FUNCTION_BLOCK PreTratamentoPreliminar (* Composite Function Block Type *)
  (* Standard: 61499-2 *)
  (* Version 0.0, 11/03/2026, template *)
  PACKAGE Hidryco.HidrycoLib;
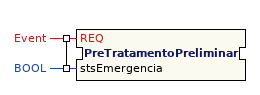
  EVENT_INPUT
    REQ WITH stsEmergencia;
  END_EVENT
  VAR_INPUT
    stsEmergencia : BOOL;
  END_VAR
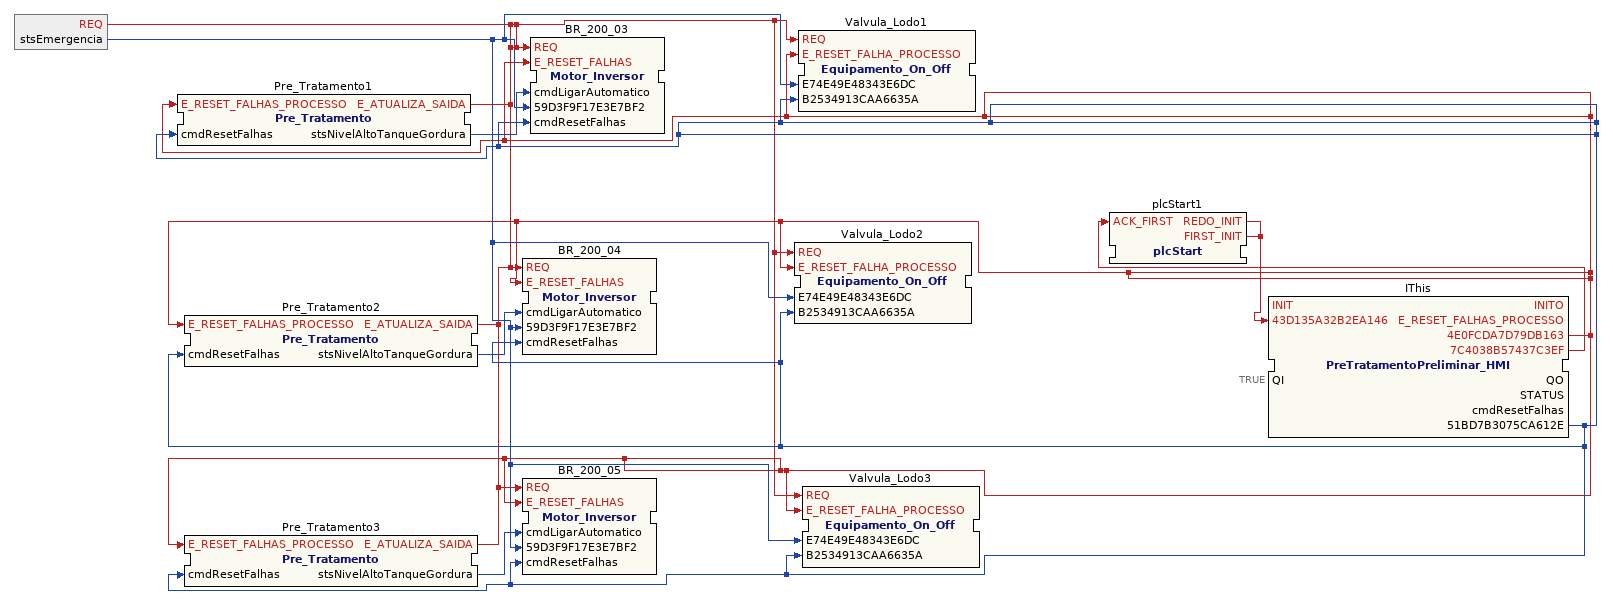
  FBS
    Pre_Tratamento1 : Pre_Tratamento;
    IThis : PreTratamentoPreliminar_HMI(QI := TRUE);
    Pre_Tratamento2 : Pre_Tratamento;
    Pre_Tratamento3 : Pre_Tratamento;
    BR_200_03 : Motor_Inversor;
    BR_200_04 : Motor_Inversor;
    BR_200_05 : Motor_Inversor;
    Valvula_Lodo1 : Equipamento_On_Off;
    Valvula_Lodo2 : Equipamento_On_Off;
    Valvula_Lodo3 : Equipamento_On_Off;
    plcStart1 : plcStart;
  END_FBS
  EVENT_CONNECTIONS
    Pre_Tratamento1.E_ATUALIZA_SAIDA TO BR_200_03.REQ;
    Pre_Tratamento2.E_ATUALIZA_SAIDA TO BR_200_04.REQ;
    Pre_Tratamento3.E_ATUALIZA_SAIDA TO BR_200_05.REQ;
    REQ TO BR_200_03.REQ;
    REQ TO Valvula_Lodo1.REQ;
    REQ TO BR_200_04.REQ;
    REQ TO Valvula_Lodo2.REQ;
    REQ TO BR_200_05.REQ;
    REQ TO Valvula_Lodo3.REQ;
    plcStart1.REDO_INIT TO IThis.43D135A32B2EA146;
    plcStart1.FIRST_INIT TO IThis.43D135A32B2EA146;
    IThis.4E0FCDA7D79DB163 TO Pre_Tratamento3.E_RESET_FALHAS_PROCESSO;
    IThis.4E0FCDA7D79DB163 TO Pre_Tratamento2.E_RESET_FALHAS_PROCESSO;
    IThis.4E0FCDA7D79DB163 TO Pre_Tratamento1.E_RESET_FALHAS_PROCESSO;
    IThis.4E0FCDA7D79DB163 TO BR_200_03.E_RESET_FALHAS;
    IThis.4E0FCDA7D79DB163 TO BR_200_04.E_RESET_FALHAS;
    IThis.4E0FCDA7D79DB163 TO BR_200_05.E_RESET_FALHAS;
    IThis.4E0FCDA7D79DB163 TO Valvula_Lodo1.E_RESET_FALHA_PROCESSO;
    IThis.4E0FCDA7D79DB163 TO Valvula_Lodo2.E_RESET_FALHA_PROCESSO;
    IThis.4E0FCDA7D79DB163 TO Valvula_Lodo3.E_RESET_FALHA_PROCESSO;
    IThis.7C4038B57437C3EF TO plcStart1.ACK_FIRST;
  END_CONNECTIONS
  DATA_CONNECTIONS
    Pre_Tratamento1.stsNivelAltoTanqueGordura TO BR_200_03.cmdLigarAutomatico;
    Pre_Tratamento2.stsNivelAltoTanqueGordura TO BR_200_04.cmdLigarAutomatico;
    Pre_Tratamento3.stsNivelAltoTanqueGordura TO BR_200_05.cmdLigarAutomatico;
    stsEmergencia TO BR_200_03.59D3F9F17E3E7BF2;
    stsEmergencia TO Valvula_Lodo1.E74E49E48343E6DC;
    stsEmergencia TO BR_200_04.59D3F9F17E3E7BF2;
    stsEmergencia TO Valvula_Lodo2.E74E49E48343E6DC;
    stsEmergencia TO BR_200_05.59D3F9F17E3E7BF2;
    stsEmergencia TO Valvula_Lodo3.E74E49E48343E6DC;
    IThis.51BD7B3075CA612E TO Pre_Tratamento3.cmdResetFalhas;
    IThis.51BD7B3075CA612E TO Pre_Tratamento2.cmdResetFalhas;
    IThis.51BD7B3075CA612E TO Pre_Tratamento1.cmdResetFalhas;
    IThis.51BD7B3075CA612E TO BR_200_05.cmdResetFalhas;
    IThis.51BD7B3075CA612E TO BR_200_04.cmdResetFalhas;
    IThis.51BD7B3075CA612E TO BR_200_03.cmdResetFalhas;
    IThis.51BD7B3075CA612E TO Valvula_Lodo3.B2534913CAA6635A;
    IThis.51BD7B3075CA612E TO Valvula_Lodo2.B2534913CAA6635A;
    IThis.51BD7B3075CA612E TO Valvula_Lodo1.B2534913CAA6635A;
  END_CONNECTIONS
END_FUNCTION_BLOCK
